// TIA Portal V18 export
// export: Created 2025-12-01T12:38:39.5147037Z, ExportSetting None, DisplayName Totally Integrated Automation Portal, DisplayVersion V18 Update 5, DisplayName TIA Portal Openness, DisplayVersion V18 Update 5, DisplayName TIA Portal Teamcenter Gateway, DisplayVersion V18, DisplayName TIA Portal Version Control Interface, DisplayVersion V18, DisplayName STEP 7 Professional, DisplayVersion V18 Update 5, DisplayName STEP 7 Safety, DisplayVersion V18, DisplayName WinCC Professional, DisplayVersion V18 Update 5
FUNCTION_BLOCK "IAI_Position"   // FB2210, LAD
{ S7_Optimized_Access := 'TRUE' }
// stored: AutoNumber false, MemoryReserve 100, SetENOAutomatically false
   VAR
      Servo5 { S7_SetPoint := 'True'} : "SevroStart&PosCheck_IAI";
      Servo6 { S7_SetPoint := 'True'} : "SevroStart&PosCheck_IAI";
      Servo7 { S7_SetPoint := 'True'} : "SevroStart&PosCheck_IAI";
   END_VAR
   VAR_TEMP
      Sevro5ActPos : Real;
      Sevro5StartList : Bool;
      Sevro6ActPos : Real;
      Sevro6StartList : Bool;
      Sevro7ActPos : Real;
      Sevro7StartList : Bool;
   END_VAR
BEGIN

REGION Network 2 (SCL)
   REGION Servo position judgment
       FOR "IAI_DeviceCtl".IAIServo[1].i := 1 TO 12 BY 1 DO
           "IAI_DeviceCtl".IAIServo[1].Pos.List["IAI_DeviceCtl".IAIServo[1].i].Pos := "IAI_A1".Auto.Pos["IAI_DeviceCtl".IAIServo[1].i].Pos;
           "IAI_DeviceCtl".IAIServo[1].Pos.List["IAI_DeviceCtl".IAIServo[1].i].Vel := "IAI_A1".Auto.Pos["IAI_DeviceCtl".IAIServo[1].i].Vel;

           "IAI_DeviceCtl".IAIServo[2].Pos.List["IAI_DeviceCtl".IAIServo[1].i].Pos := "IAI_A2".Auto.Pos["IAI_DeviceCtl".IAIServo[1].i].Pos;
           "IAI_DeviceCtl".IAIServo[2].Pos.List["IAI_DeviceCtl".IAIServo[1].i].Vel := "IAI_A2".Auto.Pos["IAI_DeviceCtl".IAIServo[1].i].Vel;

           "IAI_DeviceCtl".IAIServo[3].Pos.List["IAI_DeviceCtl".IAIServo[1].i].Pos := "IAI_A3".Auto.Pos["IAI_DeviceCtl".IAIServo[1].i].Pos;
           "IAI_DeviceCtl".IAIServo[3].Pos.List["IAI_DeviceCtl".IAIServo[1].i].Vel := "IAI_A3".Auto.Pos["IAI_DeviceCtl".IAIServo[1].i].Vel;


       END_FOR;

       (******************************************************* SV1 Z轴 ********************************************************************)
       //伺服位置判断
       #"Servo5"(iRef_Homed := 1,
                 iStandstill := FALSE,
                 iReset := "Station_Sys".Cmd.Reset,
                 interlcok := 1,
                 "iActual Posi" := "Axis_FB_DB".IAI_Axis[1].CurrentPosition,
                 "iTol+" := 0.5,
                 "iTol-" := 0.5,
                 iStartTon := T#100mS,
                 ioPoint := "IAI_DeviceCtl".IAIServo[1].Point,
                 oStartPos => #Sevro5StartList,
                 ioList := "IAI_DeviceCtl".IAIServo[1].Pos,
                 ioPosNumberSelect := "IAI_DeviceCtl".IAIServo[1].nPositionListNo);

       IF "IAI_DeviceCtl".IAIServo[1].nPositionListNo = 0 THEN
           "IAI_DeviceCtl".IAIServo[1].nPositionListNo := 1;
       END_IF;

       "Axis_FB_DB".IAI_Axis[1].Par.PosCode:="IAI_A1".Auto.Index := "IAI_DeviceCtl".IAIServo[1].nPositionListNo;

       //伺服启动
       "IAI_A1".In.iAutoStart := #Sevro5StartList AND "Station_Sys".Auto.Mode;

       (******************************************************* SV2 X轴********************************************************************)
       //伺服位置判断
       #"Servo6"(iRef_Homed := 1,
                 iStandstill := FALSE,
                 iReset := "Station_Sys".Cmd.Reset,
                 interlcok := 1,
                 "iActual Posi" := "Axis_FB_DB".IAI_Axis[2].CurrentPosition,
                 "iTol+" := 0.5,
                 "iTol-" := 0.5,
                 iStartTon := T#100mS,
                 ioPoint := "IAI_DeviceCtl".IAIServo[2].Point,
                 oStartPos => #Sevro6StartList,
                 ioList := "IAI_DeviceCtl".IAIServo[2].Pos,
                 ioPosNumberSelect := "IAI_DeviceCtl".IAIServo[2].nPositionListNo);

       IF "IAI_DeviceCtl".IAIServo[2].nPositionListNo = 0 THEN
           "IAI_DeviceCtl".IAIServo[2].nPositionListNo := 1;
       END_IF;

       "Axis_FB_DB".IAI_Axis[2].Par.PosCode:="IAI_A2".Auto.Index := "IAI_DeviceCtl".IAIServo[2].nPositionListNo;

       //伺服启动
       "IAI_A2".In.iAutoStart := #Sevro6StartList AND "Station_Sys".Auto.Mode;

       (******************************************************* SV3 Y轴********************************************************************)
       //伺服位置判断
       #"Servo7"(iRef_Homed := 1,
                 iStandstill := FALSE,
                 iReset := "Station_Sys".Cmd.Reset,
                 interlcok := 1,
                 "iActual Posi" := "Axis_FB_DB".IAI_Axis[3].CurrentPosition,
                 "iTol+" := 0.5,
                 "iTol-" := 0.5,
                 iStartTon := T#100mS,
                 ioPoint := "IAI_DeviceCtl".IAIServo[3].Point,
                 oStartPos => #Sevro7StartList,
                 ioList := "IAI_DeviceCtl".IAIServo[3].Pos,
                 ioPosNumberSelect := "IAI_DeviceCtl".IAIServo[3].nPositionListNo);

       IF "IAI_DeviceCtl".IAIServo[3].nPositionListNo = 0 THEN
           "IAI_DeviceCtl".IAIServo[3].nPositionListNo := 1;
       END_IF;

       "Axis_FB_DB".IAI_Axis[3].Par.PosCode:="IAI_A3".Auto.Index := "IAI_DeviceCtl".IAIServo[3].nPositionListNo;

       //伺服启动
       "IAI_A3".In.iAutoStart := #Sevro7StartList AND "Station_Sys".Auto.Mode;
   END_REGION
END_REGION
END_FUNCTION_BLOCK
